INTERFACE I_MutFloatArg EXTENDS I_FloatArg

PROPERTY Val : LREAL
SET
END_SET
END_PROPERTY

END_INTERFACE

(* stored: Version 1.1.0.1
   Itf I_MutFloatArg: Id {b645af79-d6f3-4181-a082-18e856162f8f}
   Property Val: Id {c833b3de-8b0f-4016-b398-0f5718568e53}
   Set Set: Id {b535739a-c7ab-4fd3-a8e9-9fed185e9628} *)
